FUNCTION_BLOCK TabletFillingControl01
VAR_INPUT
	MachineStart				:	BOOL;		// True=Machine On
	FillingPosition				:	BOOL;
	SelectTablet3				:	BOOL;		// amount (3) of tablet in tube selected 
	SelectTablet5				:	BOOL;		// amount (5) of tablet in tube selected 
	SelectTablet7				:	BOOL;		// amount (7) of tablet in tube selected 
	LightBarrier				:	BOOL;		// False = free (no tablet present)
END_VAR
VAR_OUTPUT
	BeltMotorCmdOn				:	BOOL;
	ValveCmdOpen				:	BOOL;
	LampTablet3					:	BOOL;		// True = 3 tablet in tube selected
	LampTablet5					:	BOOL;		// True = 5 tablet in tube selected
	LampTablet7					:	BOOL;		// True = 7 tablet in tube selected
END_VAR
VAR
	CountTablet3				:	CTD;		// down counter for three tablets
	CountTablet5				:	CTD;		// down counter for five tablets
	CountTablet7				:	CTD;		// down counter for seven tablets
	
	Tablet3Selected				: BOOL;
	Tablet5Selected				: BOOL;
	Tablet7Selected				: BOOL;
	FirstScan					: BOOL;
	OneShot						: BOOL;			// one shot pulse after power restart		
	srTablet3Selected			: SR;
	srTablet5Selected			: SR;
	srTablet7Selected			: SR;
	
	WAIT: SR;
	SWITCHED_ON: SR;
	WAIT_FOR_FILL_POS: SR;
	FILL_POS_REACHED: SR;
	LOAD_CTR_3_TABLETS: SR;
	LOAD_CTR_5_TABLETS: SR;
	LOAD_CTR_7_TABLETS: SR;
	
	rtCount3Tablets: R_TRIG;
	rtCount5Tablets: R_TRIG;
	rtCount7Tablets: R_TRIG;
	tonCount3Tablet: TON;
	tonCount5Tablet: TON;
	tonCount7Tablet: TON;
END_VAR
VAR // added by the converter: edge detectors and wires of the graphical bodies
    _w1 : BOOL;
END_VAR

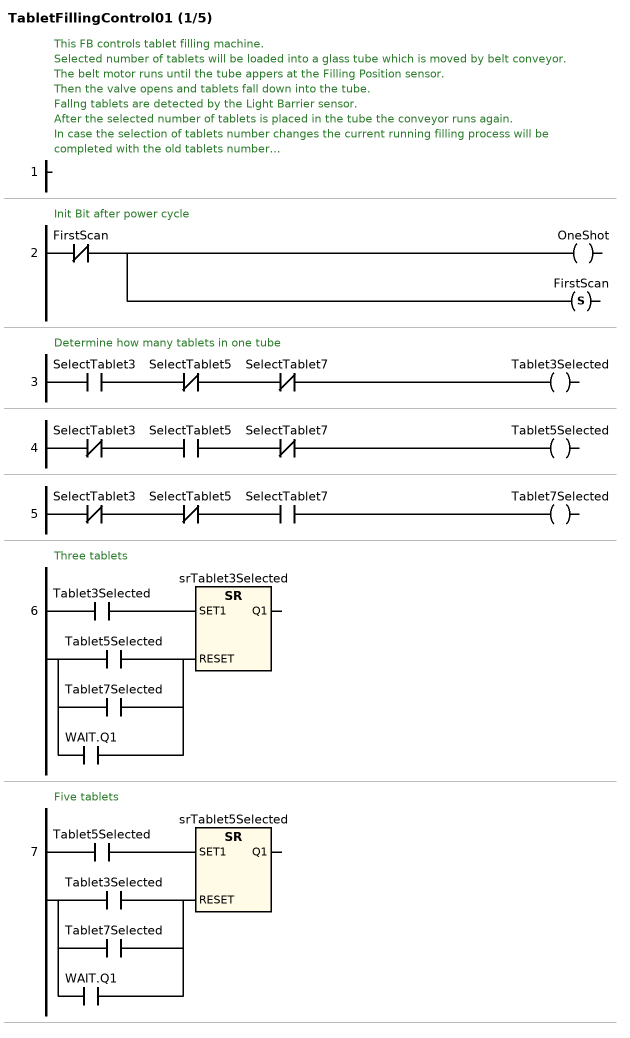
// NETWORK 1
// This FB controls tablet filling machine.
// Selected number of tablets will be loaded into a glass tube which is moved by belt conveyor.
// The belt motor runs until the tube appers at the Filling Position sensor.
// Then the valve opens and tablets fall down into the tube.
// Fallng tablets are detected by the Light Barrier sensor.
// After the selected number of tablets is placed in the tube the conveyor runs again.
// In case the selection of tablets number changes the current running filling process will be completed with the old tablets number.
// This is Version 01 of the program - only three fixed number (3,5,7) of tablets can be chosen by boolean input.

// NETWORK 2
// Init Bit after power cycle
_w1 := NOT FirstScan;
OneShot := _w1;
FirstScan S= _w1;

// NETWORK 3
// Determine how many tablets in one tube
Tablet3Selected := SelectTablet3 AND NOT SelectTablet5 AND NOT SelectTablet7;

// NETWORK 4
Tablet5Selected := NOT SelectTablet3 AND SelectTablet5 AND NOT SelectTablet7;

// NETWORK 5
Tablet7Selected := NOT SelectTablet3 AND NOT SelectTablet5 AND SelectTablet7;

// NETWORK 6
// Three tablets
srTablet3Selected(SET1 := Tablet3Selected, RESET := Tablet5Selected OR Tablet7Selected OR WAIT.Q1); // SR

// NETWORK 7
// Five tablets
srTablet5Selected(SET1 := Tablet5Selected, RESET := Tablet3Selected OR Tablet7Selected OR WAIT.Q1); // SR

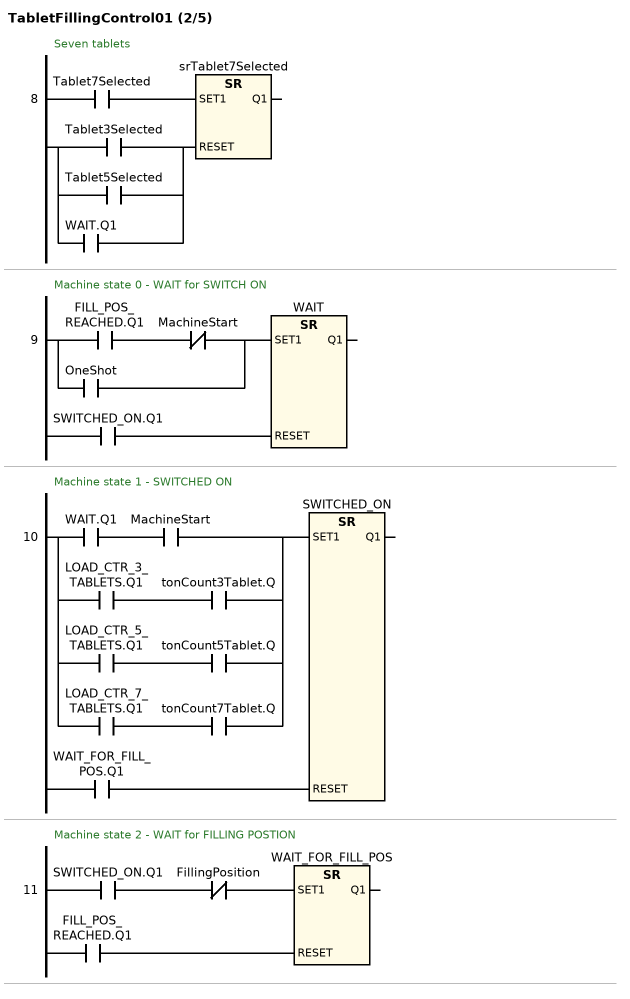
// NETWORK 8
// Seven tablets
srTablet7Selected(SET1 := Tablet7Selected, RESET := Tablet3Selected OR Tablet5Selected OR WAIT.Q1); // SR

// NETWORK 9
// Machine state 0 - WAIT for SWITCH ON
WAIT(SET1 := FILL_POS_REACHED.Q1 AND NOT MachineStart OR OneShot, RESET := SWITCHED_ON.Q1); // SR

// NETWORK 10
// Machine state 1 - SWITCHED ON
SWITCHED_ON(SET1 := WAIT.Q1 AND MachineStart OR LOAD_CTR_3_TABLETS.Q1 AND tonCount3Tablet.Q OR LOAD_CTR_5_TABLETS.Q1 AND tonCount5Tablet.Q OR LOAD_CTR_7_TABLETS.Q1 AND tonCount7Tablet.Q, RESET := WAIT_FOR_FILL_POS.Q1); // SR

// NETWORK 11
// Machine state 2 - WAIT for FILLING POSTION
WAIT_FOR_FILL_POS(SET1 := SWITCHED_ON.Q1 AND NOT FillingPosition, RESET := FILL_POS_REACHED.Q1); // SR

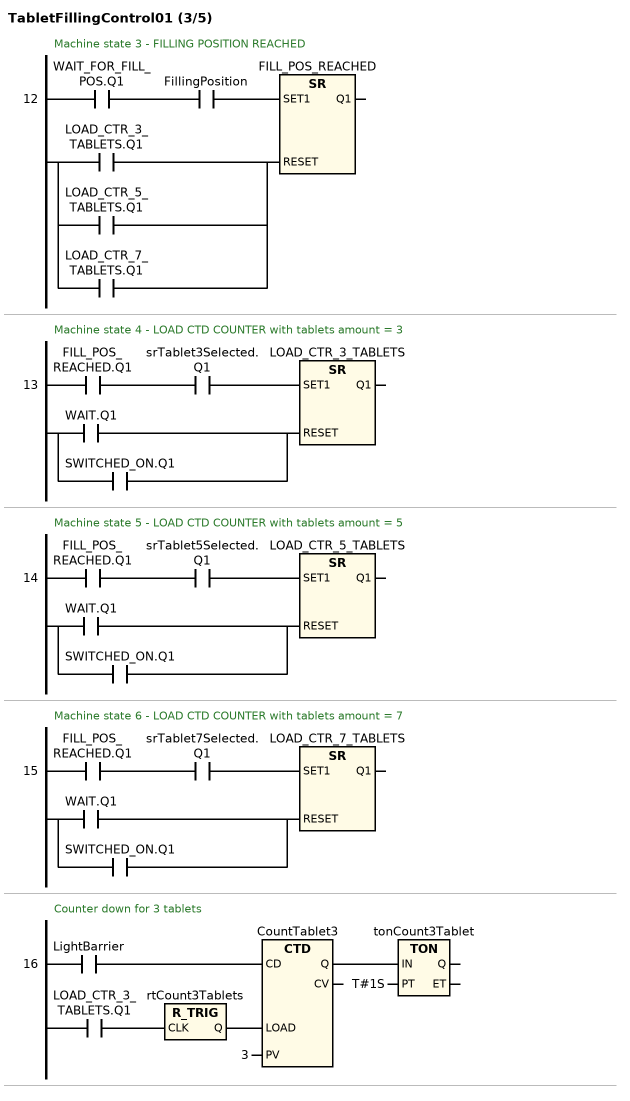
// NETWORK 12
// Machine state 3 - FILLING POSITION REACHED
FILL_POS_REACHED(SET1 := WAIT_FOR_FILL_POS.Q1 AND FillingPosition, RESET := LOAD_CTR_3_TABLETS.Q1 OR LOAD_CTR_5_TABLETS.Q1 OR LOAD_CTR_7_TABLETS.Q1); // SR

// NETWORK 13
// Machine state 4 - LOAD CTD COUNTER with tablets amount = 3
LOAD_CTR_3_TABLETS(SET1 := FILL_POS_REACHED.Q1 AND srTablet3Selected.Q1, RESET := WAIT.Q1 OR SWITCHED_ON.Q1); // SR

// NETWORK 14
// Machine state 5 - LOAD CTD COUNTER with tablets amount = 5
LOAD_CTR_5_TABLETS(SET1 := FILL_POS_REACHED.Q1 AND srTablet5Selected.Q1, RESET := WAIT.Q1 OR SWITCHED_ON.Q1); // SR

// NETWORK 15
// Machine state 6 - LOAD CTD COUNTER with tablets amount = 7
LOAD_CTR_7_TABLETS(SET1 := FILL_POS_REACHED.Q1 AND srTablet7Selected.Q1, RESET := WAIT.Q1 OR SWITCHED_ON.Q1); // SR

// NETWORK 16
// Counter down for 3 tablets
rtCount3Tablets(CLK := LOAD_CTR_3_TABLETS.Q1); // R_TRIG
CountTablet3(CD := LightBarrier, LOAD := rtCount3Tablets.Q, PV := 3); // CTD
tonCount3Tablet(IN := CountTablet3.Q, PT := T#1S); // TON

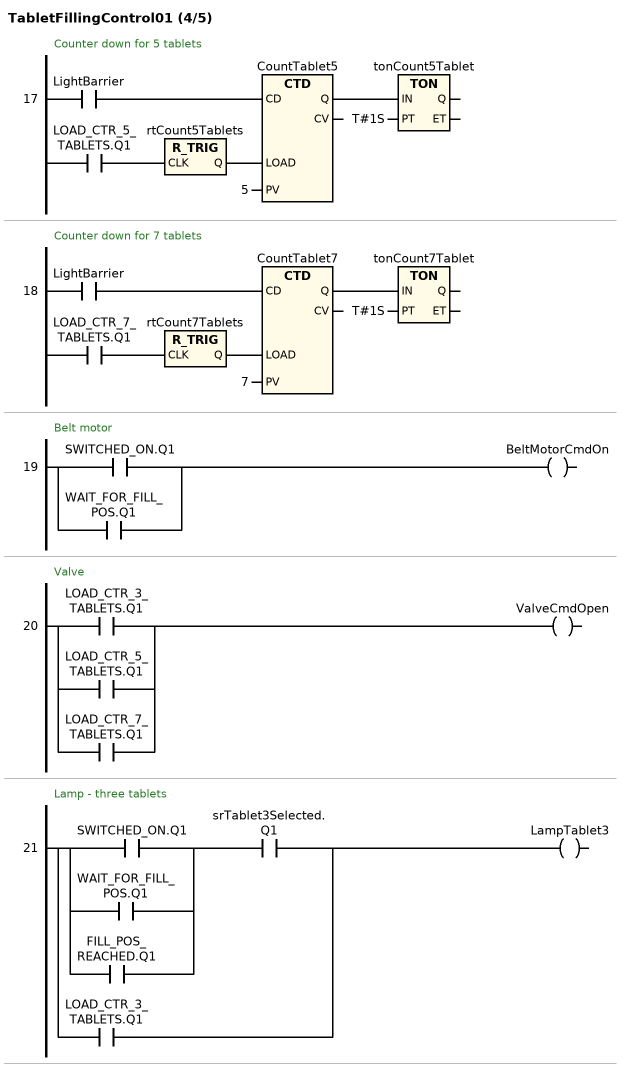
// NETWORK 17
// Counter down for 5 tablets
rtCount5Tablets(CLK := LOAD_CTR_5_TABLETS.Q1); // R_TRIG
CountTablet5(CD := LightBarrier, LOAD := rtCount5Tablets.Q, PV := 5); // CTD
tonCount5Tablet(IN := CountTablet5.Q, PT := T#1S); // TON

// NETWORK 18
// Counter down for 7 tablets
rtCount7Tablets(CLK := LOAD_CTR_7_TABLETS.Q1); // R_TRIG
CountTablet7(CD := LightBarrier, LOAD := rtCount7Tablets.Q, PV := 7); // CTD
tonCount7Tablet(IN := CountTablet7.Q, PT := T#1S); // TON

// NETWORK 19
// Belt motor
BeltMotorCmdOn := SWITCHED_ON.Q1 OR WAIT_FOR_FILL_POS.Q1;

// NETWORK 20
// Valve
ValveCmdOpen := LOAD_CTR_3_TABLETS.Q1 OR LOAD_CTR_5_TABLETS.Q1 OR LOAD_CTR_7_TABLETS.Q1;

// NETWORK 21
// Lamp - three tablets
LampTablet3 := (SWITCHED_ON.Q1 OR WAIT_FOR_FILL_POS.Q1 OR FILL_POS_REACHED.Q1) AND srTablet3Selected.Q1 OR LOAD_CTR_3_TABLETS.Q1;

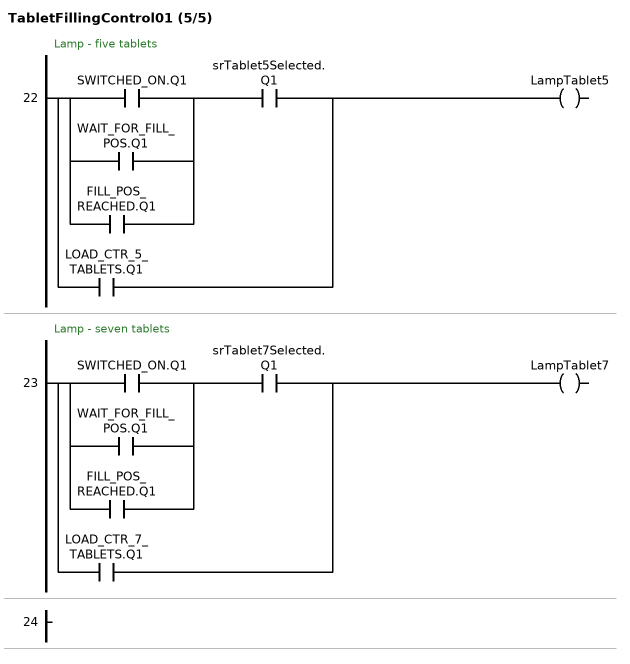
// NETWORK 22
// Lamp - five tablets
LampTablet5 := (SWITCHED_ON.Q1 OR WAIT_FOR_FILL_POS.Q1 OR FILL_POS_REACHED.Q1) AND srTablet5Selected.Q1 OR LOAD_CTR_5_TABLETS.Q1;

// NETWORK 23
// Lamp - seven tablets
LampTablet7 := (SWITCHED_ON.Q1 OR WAIT_FOR_FILL_POS.Q1 OR FILL_POS_REACHED.Q1) AND srTablet7Selected.Q1 OR LOAD_CTR_7_TABLETS.Q1;

// NETWORK 24

END_FUNCTION_BLOCK

(* stored: Version 1.1.0.1, ProductVersion 3.1.4024.15
   POU TabletFillingControl01: Id {eb71e821-67ea-47d2-a7cb-f21ac8706246}, SpecialFunc None *)
